// TIA Portal V16 export
// export: Created 2023-03-29T11:03:25.8585323Z, ExportSetting WithDefaults, DisplayName Totally Integrated Automation Portal, DisplayVersion V16 Update 6, DisplayName TIA Portal Version Control Interface, DisplayVersion V16 Update 2, DisplayName TIA Portal Openness, DisplayVersion V16 Update 6, DisplayName STEP 7 Professional, DisplayVersion V16 Update 6, DisplayName STEP 7 Safety, DisplayVersion V16, DisplayName WinCC Advanced, DisplayVersion V16 Update 6
DATA_BLOCK "CONFIG_MODBUS_TCP_SERVER"   // DB87
TITLE = CONECT MODBUS TCP SERVER
{ S7_Optimized_Access := 'TRUE' }
AUTHOR : rtecmer
VERSION : 0.1
// stored: AutoNumber true, DBAccessibleFromOPCUA true, IsOnlyStoredInLoadMemory false, IsRetainMemResEnabled false, IsWriteProtectedInAS false, MemoryReserve 100
   VAR
      CONNECT_MODBUS_TCP_Serwer_1 { S7_SetPoint := 'True'} : TCON_IP_v4;
      ERROR_STATUS_SERWER_1 : Word;   // wartość błędu
      ERROR_STATUS_SERWER_2 : Word := 16#0;   // wartość błędu
      ERROR_STATUS_SERWER_3 : Word := 16#0;   // wartość błędu
      ERROR_STATUS_SERWER_4 : Word := 16#0;   // wartość błędu
      "CONFIG SERWER_1" : Struct
         STATUS { S7_SetPoint := 'True'} : Word;   // Status połączenia TCP Modbus
         error : Bool;   // błąd
         dr : Bool;   // dane czytane
         ndr : Bool;   // dane gotowe
      END_STRUCT;
      "CONFIG SERWER_2" : Struct
         STATUS { S7_SetPoint := 'True'} : Word;   // Status połączenia TCP Modbus
         error : Bool;   // błąd
         dr : Bool;   // dane czytane
         ndr : Bool;   // dane gotowe
      END_STRUCT;
      "CONFIG SERWER_3" : Struct
         STATUS { S7_SetPoint := 'True'} : Word;   // Status połączenia TCP Modbus
         error : Bool;   // błąd
         dr : Bool;   // dane czytane
         ndr : Bool;   // dane gotowe
      END_STRUCT;
      "CONFIG SERWER_4" : Struct
         STATUS { S7_SetPoint := 'True'} : Word;   // Status połączenia TCP Modbus
         error : Bool;   // błąd
         dr : Bool;   // dane czytane
         ndr : Bool;   // dane gotowe
      END_STRUCT;
      Time_Loop_modbustcp : Time;   // czas obiegu pętli modbus tcp
   END_VAR
BEGIN
   CONNECT_MODBUS_TCP_Serwer_1.InterfaceId := 64;
   CONNECT_MODBUS_TCP_Serwer_1.ID := 1;
   CONNECT_MODBUS_TCP_Serwer_1.ConnectionType := 11;
   CONNECT_MODBUS_TCP_Serwer_1.LocalPort := 502;
END_DATA_BLOCK
